INTERFACE I_Execute EXTENDS Debug.I_Debug

METHOD Execute
VAR_INPUT
END_VAR
END_METHOD

END_INTERFACE

(* stored: Version 1.1.0.1
   Itf I_Execute: Id {a597d9f4-9133-4569-a8ee-1fffeb4f4540}
   Method Execute: Id {e865c9cb-5cde-4568-a67d-1a7697c698d2} *)
